    // Parameters for EL6 -> Serial Device
    fbSend: SendString;
    bSendBusy: BOOL;
    eLastSendErrorID: ComError_t;
    fbReceive: ReceiveString;
    sReceivedString: STRING;
    sLastReceivedString: STRING;
    bStringReceived: BOOL;
    bReceiveBusy: BOOL;
    bReceiveError: BOOL;
    eReceiveErrorID: ComError_t;
    bReceiveTimeout: BOOL;
    nReceiveCounter: UDINT;
    nSendCounter: UDINT;
    sStringToSend: STRING;
    fbFormatString: FB_FormatString;

    // Parameters for state-machine implementation
    nStep: INT := 0;
END_VAR

fbEL6Ctrl(
    Mode:= SERIALLINEMODE_EL6_22B,
    pComIn:= ADR(stIn_EL6),
    pComOut:= ADR(stOut_EL6),
    SizeComIn:= UINT_TO_INT(SIZEOF(stIn_EL6)),
    Error=> ,
    ErrorID=> eSerialLineErrorID,
    TxBuffer:= TxBuffer,
    RxBuffer:= RxBuffer );
IF fbEL6Ctrl.Error THEN
    bEL6CtrlError := TRUE;
    eEL6CtrlErrorID := fbEL6Ctrl.ErrorID;
END_IF
IF bSend THEN
    nStep := 10;
    bSend := FALSE;
    bDone := FALSE;
END_IF
// Attempt at solution that sends one command at a time, not on constant loop
CASE nStep OF
    0:
        ; // idle
    10:
        // Clear buffers in case any lingering data
        fbClearComBuffer(Buffer:=TxBuffer);
        fbClearComBuffer(Buffer:=RxBuffer);
        // Prepare string to send
        sStringToSend := CONCAT(sSendPrefix, CONCAT(sCmd, sSendSuffix));
        // Send string
        fbSend(	SendString:= sStringToSend,
                TXbuffer:= TxBuffer,
                Busy=> bSendBusy,
                Error=> eSendErrorID);
        IF fbSend.Error <> COMERROR_NOERROR THEN
            eLastSendErrorID := fbSend.Error;
        ELSE
            nSendCounter := nSendCounter + 1;
        END_IF
        nStep := nStep + 10;
    20:
        // Finish sending String
        IF fbSend.Busy THEN
            fbSend(	SendString:= sStringToSend,
                    TXbuffer:= TxBuffer,
                    Busy=> bSendBusy,
                    Error=> eSendErrorID);
            IF fbSend.Error <> COMERROR_NOERROR THEN
                eLastSendErrorID := fbSend.Error;
            ELSE
                nSendCounter := nSendCounter + 1;
            END_IF
        ELSE
            nStep := nStep + 10;
        END_IF
    30:
        // Get Reply
        fbReceive(
            Prefix:= sRecvPrefix,
            Suffix:= sRecvSuffix,
            Timeout:= tTimeout,
            ReceivedString:= sReceivedString,
            RXbuffer:= RxBuffer,
            StringReceived=> bStringReceived,
            Busy=> bReceiveBusy,
            Error=> eRecvErrorID,
            RxTimeout=> bReceiveTimeout );
        IF fbReceive.Error <> COMERROR_NOERROR THEN
            eReceiveErrorID := fbReceive.Error;
        END_IF
        IF bStringReceived THEN
            nReceiveCounter := nReceiveCounter + 1;
            // Check for response
            IF FIND(sReceivedString, sStringToSend)=0 THEN
                sResponse := sReceivedString;
                bDone := TRUE;
                nStep := 0;
            END_IF
        END_IF
END_CASE

END_FUNCTION_BLOCK

// POUs/Hardware/FB_GetPLCHostname
FUNCTION_BLOCK FB_GetPLCHostname
VAR_INPUT
    bEnable			: BOOL;
    tRetryDelay		: TIME := T#10s;
END_VAR
VAR_OUTPUT
    sHostname		: T_MaxString;
    bDone 			: BOOL;
    bError			: BOOL;
END_VAR
VAR
    fbGetHostName	: FB_GetHostName;

    tRetry 			: TON;
    bReset			: BOOL;
    bInitialized	: BOOL := FALSE;

END_VAR

IF bEnable THEN
    fbGetHostName.sNetID := '';

    IF NOT bInitialized OR (tRetry.Q AND NOT bDone) THEN
        bReset			:= TRUE;
        bInitialized	:= TRUE;
        fbGetHostName(bExecute:=FALSE);
    END_IF

    tRetry(IN:=bReset, PT:=tRetryDelay);

    bReset := FALSE;

    IF NOT bDone THEN
        fbGetHostName(bExecute:=TRUE, bError=>bError);
        IF NOT (fbGetHostName.bBusy OR bError) THEN
            sHostname	:= fbGetHostName.sHostName;
            bDone 		:= TRUE;
        END_IF
    END_IF
END_IF

END_FUNCTION_BLOCK

// POUs/Hardware/FB_GetPLCIPAddress
FUNCTION_BLOCK FB_GetPLCIPAddress
VAR_INPUT
    bEnable			: BOOL;
    tRetryDelay		: TIME := T#10s;
END_VAR
VAR_OUTPUT
    sIPAddress		: STRING(15);

    bDone 			: BOOL;
    bError			: BOOL;
END_VAR
VAR
    fbGetAdapterIP 	: FB_GetAdaptersInfo := (bExecute := TRUE, sNetID := ''); // Acquire IP of the correct adapter

    iIndex			: UDINT;

    tRetry 			: TON;
    bReset			: BOOL;
    bInitialized	: BOOL := FALSE;

END_VAR

IF bEnable THEN
    IF NOT bInitialized OR (tRetry.Q AND NOT bDone) THEN
        bReset			:= TRUE;
        bInitialized	:= TRUE;
        fbGetAdapterIP(bExecute:=FALSE);
    END_IF

    tRetry(IN:=bReset, PT:=tRetryDelay);
    bReset := FALSE;

    IF NOT bDone THEN
        fbGetAdapterIP(bExecute:=TRUE, bError=>bError);
        IF NOT (fbGetAdapterIP.bBusy or fbGetAdapterIP.bError) THEN
            FOR iIndex := 0 TO MAX_LOCAL_ADAPTERS DO
                IF FIND(fbGetAdapterIP.arrAdapters[iIndex].sIpAddr, GVL_Logger.sIpTidbit) <> 0 THEN
                    sIPAddress := fbGetAdapterIP.arrAdapters[iIndex].sIpAddr;
                    bDone := TRUE;
                    EXIT;
                END_IF
            END_FOR
        END_IF
    END_IF

END_IF

END_FUNCTION_BLOCK

// POUs/Hardware/FB_LED
FUNCTION_BLOCK FB_LED
(*
    Reads a percentage of illumination determined by the user and converts it to a raw value
    to send to the terminal output via the FB_AnalogOutput.

    The determination of the full scale raw value (FSV) is calculated via the iTermBits,
    which is setup as an input variable to be set according to the situation. This value
    is bounded by the FSV of the terminal set by the Beckhoff architecture: (2^15 - 1) = 32767.

    Through the configurable max raw value sent to the terminal output, this LED function block
    is applicable to a wider variety of hardware: whether it be simple Analog Voltage control,
    PWM voltage output, or current controlled output.

    As an initial application, this FB will be instituted for systems of vaccum chamber LED
    illuminators on TMO endstations, which are rated for 12 V max. They will be dimmed via the
    EL2502 terminal 24 V PWM output voltage control from 0-50% duty cycle.

    2022-5-03 Maarten Thomas-Bosum
*)
VAR_INPUT
    {attribute 'pytmc' := '
        pv: NAME
        io: io
        field: DESC Descriptive name for the LED
        autosave_pass0: VAL DESC
    '}
    ledName : STRING;

    iTermBits : UINT;

    {attribute 'pytmc' := '
        pv: ILL:PCT
        field: EGU %
    '}
    fIlluminatorPercent: LREAL;

    {attribute 'pytmc' := '
        pv: PWR
        field: ZNAM OFF
        field: ONAM ON
    '}
    bLedPower AT %Q*: BOOL;
END_VAR
VAR
    iIlluminatorINT AT %Q*: INT;
    fbSetIllPercent: FB_AnalogOutput;
END_VAR

// Illuminator conversion to percentage
fbSetIllPercent(
    fReal:=fIlluminatorPercent,
    fSafeMax:=100,
    fSafeMin:=0,
    iTermBits:=iTermBits,
    fTermMax:=100,
    fTermMin:=0,
    iRaw=>iIlluminatorINT);

IF  fIlluminatorPercent > 0 THEN
    bLedPower := TRUE;
ELSE
    bLEDPower := FALSE;
END_IF

END_FUNCTION_BLOCK

// POUs/Hardware/FB_TempSensor
FUNCTION_BLOCK FB_TempSensor
(*
    Handles scaling and default diagnostics for temperature sensors,
    such as thermocouples, RTDs, and others.
    2020-03-02 Zachary Lentz
*)
VAR_INPUT
    // Resolution parameter from the Beckhoff docs. Default is 0.1 for 0.1 degree resolution
    fResolution: LREAL := 0.1;
END_VAR
VAR_OUTPUT
    {attribute 'pytmc' := '
        pv: TEMP
        io: input
        field: EGU C
        field: PREC 2
    '}
    fTemp: LREAL;

    {attribute 'pytmc' := '
        pv: CONN
        io: input
        field: ONAM Connected
        field: ZNAM Disconnected
    '}
    bConnected: BOOL;

    {attribute 'pytmc' := '
        pv: ERR
        io: input
        field: ONAM True
        field: ZNAM False
    '}
    bError AT %I*: BOOL := TRUE;

    bUnderrange AT %I*: BOOL;
    bOverrange AT %I*: BOOL;
END_VAR
VAR
    iRaw AT %I*: INT;
END_VAR

// The manual states that we are disconnected if we are both overrange and in an error state
bConnected := NOT (bOverrange AND bError);
fTemp := INT_TO_LREAL(iRaw) * fResolution;

END_FUNCTION_BLOCK

// POUs/Hardware/FB_ThermoCouple
FUNCTION_BLOCK FB_ThermoCouple
(*
    Deprecated as of 2020-03-02, please use FB_TempSensor instead
    2019-10-09 Zachary Lentz
*)
{warning 'Function Block FB_ThermoCouple is deprecated and may be removed in a future release'}
VAR_INPUT
    // Ratio between raw value and actual temperature. Default is 10 for 10 steps per degree (or 0.1 degree resolution)
    iScale: INT := 10;
END_VAR
VAR_OUTPUT
    {attribute 'pytmc' := '
        pv: STC:TEMP
        io: input
    '}
    fTemp: LREAL;

    {attribute 'pytmc' := '
        pv: STC:CONN
        io: input
        field: ONAM Connected
        field: ZNAM Disconnected
    '}
    bConnected: BOOL;

    {attribute 'pytmc' := '
        pv: STC:ERR
        io: input
    '}
    bError AT %I*: BOOL;

    bUnderrange AT %I*: BOOL;
    bOverrange AT %I*: BOOL;
END_VAR
VAR
    iRaw AT %I*: INT;
END_VAR

// The manual states that we are disconnected if we are both overrange and in an error state
bConnected := NOT (bOverrange AND bError);
fTemp := INT_TO_LREAL(iRaw) / iScale;

END_FUNCTION_BLOCK

// POUs/Logger/F_SendUDPMessage
FUNCTION F_SendUDPMessage : HRESULT
VAR_INPUT
    sMessage			:	POINTER TO STRING;
    fbSocket			:	REFERENCE TO FB_ConnectionlessSocket;
    sHost				:	STRING;
    iPort				:	UINT;
END_VAR

VAR
    fbSend				:	FB_SocketUdpSendTo;
END_VAR

IF sMessage <> 0 AND __ISVALIDREF(fbSocket) THEN
    fbSend.hSocket		:= fbSocket.hSocket;
    fbSend.sRemoteHost	:= sHost;
    fbSend.nRemotePort	:= iPort;
    fbSend.pSrc 		:= sMessage;
    fbSend.cbLen		:= LEN2(sMessage);
    fbSend.bExecute	 	:= TRUE;
    fbSend();

    fbSend.bExecute 	R= fbSend.bBusy;
END_IF

END_FUNCTION

// POUs/Logger/FB_Listener
FUNCTION_BLOCK FB_Listener EXTENDS FB_ListenerBase
VAR_INPUT
END_VAR

VAR_OUTPUT
END_VAR

VAR
    nEventIdx			:	UINT := 0;
    nPendingEvents		:	UINT := 0;

    {attribute 'pytmc' := '
        pv: LogToVisualStudio
        io: io
    '}
    bLogToVisualStudio	:	BOOL := FALSE;

    {attribute 'pytmc' := '
        pv: MessagesSent
        io: i
    '}
    nCntMessagesSent 	: UDINT := 0;

    {attribute 'pytmc' := '
        pv: AlarmsRaised
        io: i
    '}
    nCntAlarmsRaised 	: UDINT := 0;

    {attribute 'pytmc' := '
        pv: AlarmsConfirmed
        io: i
    '}
    nCntAlarmsConfirmed : UDINT := 0;

    {attribute 'pytmc' := '
        pv: AlarmsCleared
        io: i
    '}
    nCntAlarmsCleared 	: UDINT := 0;

    {attribute 'pytmc' := '
        pv: MinSeverity
        io: io
    '}
    eMinSeverity	 	: TcEventSeverity;

    {attribute 'analysis' := '-33'}
    {attribute 'pytmc' := '
        pv: Log
    '}
    stEventInfo 		:	REFERENCE TO ST_LoggingEventInfo;

    stPendingEvents		:	ARRAY [0..nMaxEvents - 1] OF ST_PendingEvent;
    ipMessageConfig		:	ITcEventFilterConfig;
    fbSocket			:	POINTER TO FB_ConnectionlessSocket;
    bConfigured			:	BOOL	:= FALSE;


END_VAR

VAR_IN_OUT

END_VAR

VAR CONSTANT
    // The maximum number of events allowed *per-cycle*
    nMaxEvents			:	UINT := 10;
END_VAR

(*
    Configure an event class + severity
*)
METHOD Configure : HRESULT
VAR_INPUT
    i_EventClass 	:	GUID;
    i_MinSeverity	:	TcEventSeverity := TcEventSeverity.Verbose;
    i_fbSocket		:	POINTER TO FB_ConnectionlessSocket;
END_VAR

VAR_INST
    bSubscribed		:	BOOL := FALSE;
END_VAR
IF bSubscribed THEN
    Unsubscribe();
END_IF

THIS^.Subscribe(ADR(ipMessageConfig), 0);
bSubscribed 	:= TRUE;
eMinSeverity 	:= i_MinSeverity;
fbSocket	  	:= i_fbSocket;

IF (ipMessageConfig = 0) THEN
    Configure 	:= 1;
    bConfigured := FALSE;
ELSE
    ipMessageConfig.AddEventClass(i_EventClass, i_MinSeverity);
    Configure 	:= 0;
    bConfigured := TRUE;
END_IF
END_METHOD

{attribute 'analysis' := '-33'}
PROPERTY PUBLIC LogToVisualStudio : BOOL
GET
LogToVisualStudio := bLogToVisualStudio;
END_GET
SET
VAR
    bValue : BOOL;
END_VAR
THIS^.bLogToVisualStudio := bValue;
END_SET
END_PROPERTY

METHOD OnAlarmCleared
VAR_INPUT
    fbEvent : REFERENCE TO FB_TcEvent;
END_VAR
(* Callback run from THIS^.Execute() *)
nCntAlarmsCleared := nCntAlarmsCleared + 1;
StoreEvent(fbEvent, eEventType:=E_LogEventType.AlarmCleared);
END_METHOD

METHOD OnAlarmConfirmed
VAR_INPUT
    fbEvent : REFERENCE TO FB_TcEvent;
END_VAR
(* Callback run from THIS^.Execute() *)
nCntAlarmsConfirmed := nCntAlarmsConfirmed + 1;
StoreEvent(fbEvent, eEventType:=E_LogEventType.AlarmConfirmed);
END_METHOD

METHOD OnAlarmRaised
VAR_INPUT
    fbEvent : REFERENCE TO FB_TcEvent;
END_VAR
(* Callback run from THIS^.Execute() *)
nCntAlarmsRaised := nCntAlarmsRaised + 1;
StoreEvent(fbEvent, eEventType:=E_LogEventType.AlarmRaised);
END_METHOD

METHOD OnMessageSent
VAR_INPUT
    fbEvent : REFERENCE TO FB_TcEvent;
END_VAR
(* Callback run from THIS^.Execute() *)
nCntMessagesSent := nCntMessagesSent + 1;
StoreEvent(fbEvent, eEventType:=E_LogEventType.MessageSent);
END_METHOD

METHOD PublishEvents : HRESULT
VAR
    nEvent				:	UINT;
    stPendingEvent		:	REFERENCE TO ST_PendingEvent;
    stEventInfo			:	REFERENCE TO ST_LoggingEventInfo;
    fbRequestEventText	:	REFERENCE TO FB_RequestEventText;
END_VAR

VAR_INST
    fbJson				:	FB_JsonSaxWriter;
    fbJsonDataType		:	FB_JsonReadWriteDataType;
    sJsonDoc			:	STRING(10000);

END_VAR

IF nPendingEvents = 0 THEN
    RETURN;
END_IF

FOR nEvent := 0 TO nMaxEvents - 1 DO
    stPendingEvent REF= stPendingEvents[nEvent];
    IF NOT stPendingEvent.bInUse THEN
        CONTINUE;
    END_IF

    fbRequestEventText REF= stPendingEvent.fbRequestEventText;
    stEventInfo 	   REF= stPendingEvent.stEventInfo;

    IF fbRequestEventText.bError THEN
        stEventInfo.Msg := '(Unable to retrieve message)';
    ELSIF NOT fbRequestEventText.bBusy THEN
        fbRequestEventText.GetString(stEventInfo.msg, SIZEOF(stEventInfo.msg));
    ELSE
        CONTINUE;
    END_IF

    IF bConfigured THEN
        stEventInfo.plc := GVL_Logger.sPlcHostname;

        // Generate the JSON message
        fbJson.ResetDocument();
        fbJsonDataType.AddJsonValueFromSymbol(fbJson, 'ST_LoggingEventInfo', SIZEOF(stEventInfo), ADR(stEventInfo));
        fbJson.CopyDocument(sJsonDoc, SIZEOF(sJsonDoc));

        SendMessage(sMessage:=ADR(sJsonDoc));
    END_IF

    // Mark as not in use, and fill in this event in the next StoreEvent call
    nPendingEvents			:= nPendingEvents - 1;
    stPendingEvent.bInUse 	:= FALSE;
    nEventIdx 				:= nEvent;

END_FOR
END_METHOD

METHOD SendMessage : HRESULT
VAR_INPUT
    sMessage		:	POINTER TO STRING;
END_VAR

VAR
    sLogStr			:	T_MaxString;
END_VAR
(* For subclasses to override, if necessary *)
IF sMessage = 0 THEN
    RETURN;
END_IF

// Optionally log it to Visual Studio's message list
IF bLogToVisualStudio THEN
     // Keep the message length under 255 (extended string function for LEFT/MID do not exist)
    STRNCPY(ADR(sLogStr), sMessage, MIN(220, SIZEOF(sLogStr)));
    ADSLOGSTR(
        msgCtrlMask := ADSLOG_MSGTYPE_HINT,
        msgFmtStr   := '[Logger JSON Debug] %s',
        strArg      := sLogStr
    );
END_IF

IF fbSocket <> 0 THEN
    // And send it along to logstash
    F_SendUDPMessage(sMessage:=sMessage, fbSocket:=fbSocket^,
                     sHost:=GVL_Logger.cLogHost, iPort:=GVL_Logger.iLogPort);
END_IF
END_METHOD

METHOD PRIVATE StoreEvent : HRESULT
VAR_INPUT
    fbEvent		:	REFERENCE TO FB_TcEvent;
    eEventType	:	E_LogEventType;
END_VAR

VAR
    stPendingEvent	:	REFERENCE TO ST_PendingEvent;
    stEventInfo		:	REFERENCE TO ST_LoggingEventInfo;
    nFailures		:	UINT := 0;
END_VAR
IF fbEvent.eSeverity < eMinSeverity THEN
    // Ignore all messages below the minimum severity
    RETURN;
ELSIF NOT __ISVALIDREF(fbEvent) THEN
    RETURN;
END_IF

// Find the next slot to use in stPendingEvents
WHILE stPendingEvents[nEventIdx].bInUse AND nFailures < nMaxEvents DO
    nFailures := nFailures + 1;
    IF ((nEventIdx := (nEventIdx + 1)) = nMaxEvents) THEN
        nEventIdx := 0;
    END_IF
END_WHILE

IF (nFailures = nMaxEvents) THEN
    ADSLOGSTR(
        msgCtrlMask := ADSLOG_MSGTYPE_ERROR,
        msgFmtStr   := 'Logging message buffer full (%s)',
        strArg		:= UINT_TO_STRING(nMaxEvents),
    );
    RETURN;
END_IF

nPendingEvents			:=	nPendingEvents + 1;
nCntMessagesSent 		:=	nCntMessagesSent + 1;

stPendingEvent			REF= stPendingEvents[nEventIdx];
stEventInfo 			REF= stPendingEvent.stEventInfo;
stPendingEvent.bInUse 	:= TRUE;

stEventInfo.id 			:= fbEvent.nEventId;
stEventInfo.event_class	:= GUID_TO_STRING(fbEvent.EventClass);
stEventInfo.severity 	:= fbEvent.eSeverity;
stEventInfo.ts			:= F_ConvertTicksToUnixTimestamp(fbEvent.nTimestamp);
stEventInfo.source 		:= fbEvent.ipSourceInfo.sName;
stEventInfo.event_type	:= eEventType;

fbEvent.GetJsonAttribute(stEventInfo.json, SIZEOF(stEventInfo.json));
stPendingEvent.fbRequestEventText.Request(eventClass:=fbEvent.EventClass, nEventId:=fbEvent.nEventId, nLangId:=1033, ipArgs:=fbEvent.ipArguments);
END_METHOD

END_FUNCTION_BLOCK

// POUs/Logger/FB_LogHandler
FUNCTION_BLOCK FB_LogHandler
VAR_INPUT

    {attribute 'pytmc' := '
        pv: ADS
    '}
    fbTcAdsListener : FB_Listener;

    {attribute 'pytmc' := '
        pv: Router
    '}
    fbTcRouterListener : FB_Listener;

    {attribute 'pytmc' := '
        pv: RTime
    '}
    fbTcRTimeListener : FB_Listener;

    {attribute 'pytmc' := '
        pv: System
    '}
    fbTcSystemListener : FB_Listener;

    {attribute 'pytmc' := '
        pv: Windows
    '}
    fbWindowsListener : FB_Listener;

    {attribute 'pytmc' := '
        pv: LCLS
    '}
    fbLCLSListener 	: FB_Listener;

END_VAR
VAR_OUTPUT
END_VAR

VAR

    bInitialized	:	BOOL	:= FALSE;
    bReadyToLog		: 	BOOL	:= FALSE;
    rtFirstLog		: 	R_TRIG;

    fbGetHostName 	: FB_GetPLCHostname;
    fbGetIP		 	: FB_GetPLCIPAddress;

    fbListener		:	REFERENCE TO FB_Listener;
    fbListeners		: 	ARRAY [0..nNumListeners - 1] OF POINTER TO FB_Listener;

    // Default minimum severity for subscriptions
    eMinSeverity	:	TcEventSeverity := TcEventSeverity.Verbose;

    {attribute 'naming' := 'omit'}
    rtReset				:	R_TRIG; //Reset trigger
    bReset				:	BOOL;

    fbSocket	   		:	FB_ConnectionlessSocket;

    nI					:	UINT;

    SocketEnable : BOOL;

    ctuSocketError : CTU := (PV:=3); // Circuit breaker for socket errors. 3 errors before it stops.

    tRetryConnection : TON := (PT:=T#1h); // Retry after an hour

    tofTrickleBreakerPre : TOF := (PT:=T#1s);
    tonTrickleBreaker : TON := (PT := GVL_Logger.nTrickleTripTime);
    bTripCon : BOOL;
END_VAR

VAR CONSTANT
    nNumListeners		:	UINT	:= 6;
END_VAR

IF NOT bInitialized THEN
    bInitialized := TRUE;
    fbTcAdsListener.Configure(i_EventClass:=TC_EVENT_CLASSES.TcGeneralAdsEventClass, i_MinSeverity:=eMinSeverity, i_fbSocket:=ADR(fbSocket));
    fbTcRouterListener.Configure(i_EventClass:=TC_EVENT_CLASSES.TcRouterEventClass, i_MinSeverity:=eMinSeverity, i_fbSocket:=ADR(fbSocket));
    fbTcRTimeListener.Configure(i_EventClass:=TC_EVENT_CLASSES.TcRTimeEventClass, i_MinSeverity:=eMinSeverity, i_fbSocket:=ADR(fbSocket));
    fbTcSystemListener.Configure(i_EventClass:=TC_EVENT_CLASSES.TcSystemEventClass, i_MinSeverity:=eMinSeverity, i_fbSocket:=ADR(fbSocket));
    fbWindowsListener.Configure(i_EventClass:=TC_EVENT_CLASSES.Win32EventClass, i_MinSeverity:=eMinSeverity, i_fbSocket:=ADR(fbSocket));
    fbLCLSListener.Configure(i_EventClass:=TC_EVENT_CLASSES.LCLSGeneralEventClass, i_MinSeverity:=eMinSeverity, i_fbSocket:=ADR(fbSocket));

    fbListeners[0] := ADR(fbTcAdsListener);
    fbListeners[1] := ADR(fbTcRouterListener);
    fbListeners[2] := ADR(fbTcRTimeListener);
    fbListeners[3] := ADR(fbTcSystemListener);
    fbListeners[4] := ADR(fbWindowsListener);
    fbListeners[5] := ADR(fbLCLSListener);

END_IF

fbGetHostName(
    bEnable := TRUE,
    sHostname => GVL_Logger.sPlcHostname,
);

fbGetIP(
    bEnable := TRUE,
    sIPAddress => fbSocket.sLocalHost
);

(* Ensure the socket is ready for when JSON documents are emitted *)
rtReset(CLK:=bReset);

IF (rtReset.Q AND fbSocket.bEnable) THEN
    fbSocket(bEnable:=FALSE);
END_IF

// Disable fbSocket if too many errors occur
ctuSocketError(CU:=fbSocket.bError, RESET:=tRetryConnection.Q OR rtReset.Q);
SocketEnable R= ctuSocketError.Q;
// Retry an hour later
tRetryConnection(IN:=ctuSocketError.Q);
SocketEnable S= tRetryConnection.Q OR rtReset.Q;

fbSocket(
    nLocalPort:=0,
    bEnable:=fbGetIP.bDone,
    nMode:=CONNECT_MODE_ENABLEDBG,
);

bReadyToLog := (
    fbGetHostName.bDone AND
    fbGetIP.bDone AND
    bInitialized AND
    fbSocket.bEnable AND
    NOT fbSocket.bError AND
    fbSocket.eState = E_SocketConnectionlessState.eSOCKET_CREATED
);
rtFirstLog(CLK:=bReadyToLog);

IF rtFirstLog.Q THEN
    fbRootLogger(sMsg:='Logging system online', eSevr:=TcEventSeverity.Info,
                 eSubsystem:=E_Subsystem.NILVALUE);
END_IF

CircuitBreaker();

(* Poke all of the listeners *)
FOR nI := 0 TO nNumListeners - 1 DO
    fbListener REF= fbListeners[nI]^;
    fbListener.Execute();
    fbListener.PublishEvents();
END_FOR

ACTION CircuitBreaker:
// Global log circuit breaker
(*
Logic explanation
We want to trip if there is a constant stream of messages being emitted by this PLC. We also
only want the noisy offenders to trip. To target them we set a global trickle tripped flag
using this logic here. Then each individual FB_LogMessage evaluates itself to see if it's
sending a message too frequently (ie. it's being called to often).

This logic is attempting to implement the following:
1. Trip if the total events exceeds the nTrickleThreshold for >10s
2. Sustain the timer if the event count drops for a handful of cycles since usually a cycle amounts to 10ms, losing a few
should not stop the trickle timer.
*)
bTripCon := GVL_Logger.nGlobAccEvents >0;

tofTrickleBreakerPre(IN:=bTripCon);
tonTrickleBreaker(IN:=tofTrickleBreakerPre.Q);

GVL_Logger.bTrickleTripped S= tonTrickleBreaker.Q AND bTripCon;

GVL_Logger.nGlobAccEvents := 0; // reset the count for the next cycle
END_ACTION

END_FUNCTION_BLOCK

// POUs/Logger/SYSTEM_TIME_TO_RFC3339
//Converts Beckhoff PLC SYSTEMTIME to RFC3339 time format as a string
{attribute 'naming' := 'omit'}
{attribute 'analysis' := '-23'}
FUNCTION SYSTEM_TIME_TO_RFC3339 : STRING(255)
VAR_INPUT
    {attribute 'naming' := 'omit'}
    tCurrentTime	:	TIMESTRUCT; //TIMESTRUCT Time to convert to RFC3339
END_VAR
VAR
END_VAR

SYSTEM_TIME_TO_RFC3339 := CONCAT(REPLACE(SYSTEMTIME_TO_STRING(tCurrentTime), 'T', 1, 11), 'Z');

END_FUNCTION

// POUs/Tests/FB_CircuitBreaker_Test
{attribute 'call_after_init'}
FUNCTION_BLOCK FB_CircuitBreaker_Test EXTENDS TcUnit.FB_TestSuite
VAR_INPUT
END_VAR
VAR_OUTPUT
END_VAR
VAR
END_VAR

AutoReset();
SingleBadLogger();
DeathByManySmall();

METHOD AutoReset
VAR_INPUT
END_VAR
VAR_INST
    fbLog : FB_LogMessage := (
        bEnableAutoReset:=TRUE,
        nTripResetPeriod := T#5s);

    //Auto reset test
    tonAutoResetTest : TON;

    {attribute 'analysis' := '-27'}
    Init : BOOL := TRUE;
END_VAR
(* Test that the CB resets itself after a cooldown period *)
TEST('AutoReset');
IF Init THEN
    fbLog.CircuitBreaker();
    WRITE_PROTECTED_BOOL(ADR(fbLog.bTripped), TRUE);
    WRITE_PROTECTED_BOOL(ADR(fbLog.bLocalTripped), TRUE);
    fbLog.CircuitBreaker();
    fbLog.CircuitBreaker();
    Init := FALSE;
END_IF

tonAutoResetTest(IN:=NOT Init, PT:=T#6s);

IF tonAutoResetTest.Q THEN

    fbLog.CircuitBreaker();

    AssertFalse(fbLog.bTripped,
        'Circuit breaker should be reset automatically');

    TEST_FINISHED_NAMED('AutoReset');
END_IF
END_METHOD

METHOD DeathByManySmall
VAR_INPUT
END_VAR
VAR

END_VAR
VAR_INST
    fbLogNoisy : FB_LogMessage;
    tNoisy : TON := (PT:=T#50ms); //50ms is > the local trip threshold default of 1ms
    fbLogNice : FB_LogMessage := (nTrickleTripThreshold:=T#2s);
    tNice : TON := (PT:=T#5s);
    tTrickle : TON := (PT:= GVL_Logger.nTrickleTripTime + T#1s);
    fbLogHandler : FB_LogHandler;
END_VAR
TEST('ManySmall');
// Create a condition where
// a few loggers did their thing, while keeping under the
// local logging rate limit until the global trickle trip
// was triggered. Then verify only those loggers that
// were just a little too noisy, would trip off, while others stayed up.

fbLogHandler.CircuitBreaker();

// Call this guy every 50ms or so.
tNoisy(IN := NOT tNoisy.Q);
IF tNoisy.Q THEN
    fbLogNoisy.CircuitBreaker();
END_IF

// Call this guy every 5s or so
tNice(IN := NOT tNoisy.Q);
IF tNice.Q THEN
    fbLogNice.CircuitBreaker();
END_IF

tTrickle(IN:=TRUE);
IF tTrickle.Q THEN
    AssertTrue(fbLogNoisy.bLocalTrickleTripped AND NOT fbLogNice.bLocalTrickleTripped,
            'Only Noisy should be tripped.');
    TEST_FINISHED_NAMED('ManySmall');
END_IF
END_METHOD

METHOD SingleBadLogger
VAR_INPUT
END_VAR
VAR
    idx : UINT;
END_VAR
VAR_INST
    fbLog : FB_LogMessage := (
        bEnableAutoReset:=TRUE,
        nTripResetPeriod := T#5s);
END_VAR
ResetCircuitBreakerGlobals();

(* In this scenario, a logger trips off because it has been called too many times
in one cycle, leading to a large excess of messages.
*)
TEST('LocalFastTrip');
    FOR idx := 0 TO GVL_LOGGER.nMinTimeViolationAcceptable + 1 DO
        fbLog.CircuitBreaker();
    END_FOR

    AssertTrue(fbLog.bLocalTripped AND NOT fbLog.bLocalTrickleTripped,
        'Only local trip should occur in these conditions');
TEST_FINISHED();
END_METHOD

END_FUNCTION_BLOCK

// POUs/Tests/ResetCircuitBreakerGlobals
FUNCTION ResetCircuitBreakerGlobals : BOOL
VAR_INPUT
END_VAR
VAR
END_VAR

GVL_Logger.bTrickleTripped := FALSE;
GVL_Logger.nGlobAccEvents := 0;

END_FUNCTION

// POUs/Tests/FB_ECATAutoRestart_Test

FUNCTION_BLOCK FB_ECATAutoRestart_Test EXTENDS TcUnit.FB_TestSuite
VAR
    fbECATAutoRestart : FB_ECATAutoRestart;

    fbTON_TestTimer		: TON;
    bStartTest			: BOOL := FALSE;


END_VAR


TestSingleLogPerTransitionExpect4Logs();
TestAnyStateExpectChangeToOpStateInSeq();
TestNotEnabledExpectNoStateChange();
Test5RetriesExpectErrorStopTrying();
TestBadAddressExpectError();


METHOD Test5RetriesExpectErrorStopTrying
VAR_INPUT
END_VAR
VAR
    nIndex                  : INT;
    nStateMachineState      : INT;

    // State Machine Control Inputs
    bEnable                 : BOOL;
    bfbGetBusy              : BOOL;
    bfbGetError              : BOOL;
    nCurretState            : WORD;
    bfbSetBusy              : BOOL;
    bfbSetError             : BOOL;

    // State Machine Control Outputs
    bfbGetUpdatedState      : BOOL;
    bSetNextState           : BOOL;
    nNextState              : WORD;
    sLogMessage             : T_MaxString;
    bLog                    : BOOL;

END_VAR

TEST('Test5RetriesExpectErrorStopTrying');

nStateMachineState := 1; // Start Test on Start State
bEnable := TRUE;
bfbGetBusy := FALSE;
bfbGetError := FALSE;
nCurretState := EC_DEVICE_STATE_PREOP;
bfbSetBusy := FALSE;
bfbSetError := TRUE;

FOR nIndex := 1 TO 20 DO
    fbECATAutoRestart.StateMachine(bEnable:=bEnable,
        bfbGetBusy := bfbGetBusy,
        bfbGetError := bfbGetError,
        bfbGetUpdatedState => bfbGetUpdatedState,
        nCurretState := nCurretState,
        nNextState => nNextState,
        sLogMessage=> sLogMessage,
        bLog=> bLog,
        bSetNextState=> bSetNextState,
        bfbSetBusy := bfbSetBusy,
        bfbSetError := bfbSetError);
END_FOR


AssertEquals_BOOL(Expected:=TRUE,
                    Actual:= fbECATAutoRestart.bStopTrying,
                    Message:='bStopTrying was not set after trying to get new position after 20 Cycles');

// CLEAR ANY ERRORS AFTER TESTS
FOR nIndex := 1 TO 3 DO
    fbECATAutoRestart.StateMachine(bEnable:=FALSE,
        bfbGetBusy := bfbGetBusy,
        bfbGetError := bfbGetError,
        bfbGetUpdatedState => bfbGetUpdatedState,
        nCurretState := nCurretState,
        nNextState => nNextState,
        sLogMessage=> sLogMessage,
        bLog=> bLog,
        bSetNextState=> bSetNextState,
        bfbSetBusy := bfbSetBusy,
        bfbSetError := bfbSetError);
END_FOR

TEST_FINISHED();
END_METHOD


METHOD TestAnyStateExpectChangeToOpStateInSeq
VAR_INPUT
END_VAR
VAR

    // State Machine Control Inputs
    bEnable                 : BOOL;
    bfbGetBusy              : BOOL;
    bfbGetError				: BOOL;
    nCurretState            : WORD;
    bfbSetBusy              : BOOL;
    bfbSetError             : BOOL;

    // State Machine Control Outputs
    bfbGetUpdatedState      : BOOL;
    bSetNextState           : BOOL;
    nNextState              : WORD;
    sLogMessage             : T_MaxString;
    bLog                    : BOOL;
    // TestAnyStateChangeOpInSeq Vars

    nIndex          : INT := 1;
    aPossibleStart : ARRAY [1 .. 4] OF BYTE := [EC_DEVICE_STATE_BOOTSTRAP,
                                                EC_DEVICE_STATE_INIT,
                                                EC_DEVICE_STATE_PREOP,
                                                EC_DEVICE_STATE_SAFEOP];
    nStartIndex : INT := 0;


END_VAR

TEST('TestAnyStateExpectChangeToOpStateInSeq');


bEnable := TRUE;
bfbGetBusy := FALSE;
bfbSetBusy := FALSE;
bfbSetError := FALSE;
bfbGetError := FALSE;




FOR nStartIndex := 1 TO 4 DO
    nCurretState := aPossibleStart[nStartIndex];
    // Takes 3 cycles for statemachine to update state
    // 4 - nStartIndex is number of steps needed to return to OP
    FOR nIndex := 1 TO 3 * 4 - nStartIndex DO
    fbECATAutoRestart.StateMachine
            (bEnable:=bEnable,
            bfbGetBusy := bfbGetBusy,
            bfbGetError := bfbGetError,
            bfbGetUpdatedState => bfbGetUpdatedState,
            nCurretState := nCurretState,
            nNextState => nNextState,
            sLogMessage=> sLogMessage,
            bLog=> bLog,
            bSetNextState=> bSetNextState,
            bfbSetBusy := bfbSetBusy,
            bfbSetError := bfbSetError);

    IF bSetNextState THEN
        nCurretState := nNextState;
    END_IF
    END_FOR

    AssertEquals_BYTE(Expected:=EC_DEVICE_STATE_OP,
        Actual:= TO_BYTE(nCurretState),
        Message:='Test Did not Return to OP');
END_FOR

 TEST_FINISHED();
END_METHOD


METHOD TestBadAddressExpectError
VAR_INPUT
END_VAR
VAR
    bError				: BOOL;
    bErrorId			: UDINT;
    nIndex				: INT;
END_VAR

TEST('TestBadAddressExpectError');

FOR nIndex := 1 TO 6 DO

    fbECATAutoRestart(sNetId:='1.0.0.0.1',
                    nSlaveAddr:=11101,
                    bEnable:= TRUE,
                    bError=>bError,
                    nErrorId=>bErrorId);


    IF bError THEN
    AssertEquals_BOOL(Expected:=TRUE,
        Actual:=bError,
        Message:= 'Expected bError to be TRUE');

    AssertEquals_UDINT(Expected:= 7,
        Actual:= bErrorId,
        Message:= 'Expected ERR_TARGETMACHINENOTFOUND (0x7)');

    END_IF
END_FOR

   TEST_FINISHED();
END_METHOD


METHOD TestNotEnabledExpectNoStateChange
VAR_INPUT
END_VAR
VAR
    nStateMachineStartState      : INT;
    // State Machine Control Inputs
    bEnable                 : BOOL;
    bfbGetBusy              : BOOL;
    bfbGetError				: BOOL;
    nCurretState            : WORD;
    bfbSetBusy              : BOOL;
    bfbSetError             : BOOL;

    // State Machine Control Outputs
    bfbGetUpdatedState      : BOOL;
    bSetNextState           : BOOL;
    nNextState              : WORD;
    sLogMessage             : T_MaxString;
    bLog                    : BOOL;

END_VAR

TEST('TestNotEnabledExpectNoStateChange');

nStateMachineStartState := 1;
bEnable := FALSE;
bfbGetBusy := FALSE;
nCurretState := EC_DEVICE_STATE_PREOP;
bfbSetBusy := FALSE;
bfbSetError := TRUE;
bfbGetError := FALSE;

fbECATAutoRestart.StateMachine(bEnable:=bEnable,
    bfbGetBusy := bfbGetBusy,
    bfbGetError	:= bfbGetError,
    bfbGetUpdatedState => bfbGetUpdatedState,
    nCurretState := nCurretState,
    nNextState => nNextState,
    sLogMessage=> sLogMessage,
    bLog=> bLog,
    bSetNextState=> bSetNextState,
    bfbSetBusy := bfbSetBusy,
    bfbSetError := bfbSetError);


AssertEquals_WORD(Expected:= 0,
                    Actual:= nNextState,
                    Message:= 'When bEnable is False, nNextState should not return anything');

TEST_FINISHED();
END_METHOD

METHOD TestSingleLogPerTransitionExpect4Logs
VAR_INPUT
END_VAR

VAR
        // State Machine Control Inputs
    bEnable                 : BOOL;
    bfbGetBusy              : BOOL;
    nCurretState            : WORD;
    bfbSetBusy              : BOOL;
    bfbSetError             : BOOL;
    bfbGetError				: BOOL;

    // State Machine Control Outputs
    bfbGetUpdatedState      : BOOL;
    bSetNextState           : BOOL;
    nNextState              : WORD;
    sLogMessage             : T_MaxString;
    bLog                    : BOOL;

    nIndex          : INT := 1;
    nLogCount       : INT := 0;
END_VAR

TEST('TestSingleLogPerTransitionExpect4Logs');

fbTON_TestTimer(IN:=bStartTest,PT:=T#1s);
IF  NOT bStartTest THEN bStartTest := TRUE; END_IF

bEnable := TRUE;
bfbGetBusy := FALSE;
bfbSetBusy := FALSE;
bfbSetError := FALSE;
bfbGetError := FALSE;

nCurretState := EC_DEVICE_STATE_INIT;
// Using More cyles then needed
 FOR nIndex := 1 TO 3 * 4 DO
    fbECATAutoRestart.StateMachine
            (bEnable:=bEnable,
            bfbGetBusy := bfbGetBusy,
            bfbGetError := bfbGetError,
            bfbGetUpdatedState => bfbGetUpdatedState,
            nCurretState := nCurretState,
            nNextState => nNextState,
            sLogMessage=> sLogMessage,
            bLog=> bLog,
            bSetNextState=> bSetNextState,
            bfbSetBusy := bfbSetBusy,
            bfbSetError := bfbSetError);

    IF bLog THEN
        nLogCount := nLogCount + 1;
    END_IF
END_FOR

AssertEquals_INT(Expected:= 4,
    Actual:=nLogCount,
    Message:='More than 4 Logs where Produced');

TEST_FINISHED();
END_METHOD

END_FUNCTION_BLOCK

// POUs/Tests/FB_FlutterDetection_Test
FUNCTION_BLOCK FB_FlutterDetection_Test EXTENDS TcUnit.FB_TestSuite
VAR_INPUT
END_VAR
VAR_OUTPUT
END_VAR
VAR
    fbFlutterDet : FB_FlutterDetection;

    nFirstCycleCount : UDINT;
    nCurrentSystemCycle : UDINT;
    nCurrentLocalCycle : UDINT;
END_VAR

TestFlutterResolution();
TestFlutterReset();

METHOD TestFlutterReset
VAR_INST
    fbTestTimer : TON := (PT := T#300ms);
    bInit : BOOL := FALSE;
    bVarToMonitor : BOOL := TRUE;
END_VAR
(* after trip, function should latch exceeded flag remains tripped. Finally,
check that after reset, the coount resets and the exceeded flag
goes low, then trips again. *)
TEST('TestFlutterReset');
IF NOT bInit THEN
    nFirstCycleCount := _TaskInfo[GETCURTASKINDEXEX()].CycleCount;
    bInit := TRUE;
END_IF
nCurrentSystemCycle := _TaskInfo[GETCURTASKINDEXEX()].CycleCount;
nCurrentLocalCycle := nCurrentSystemCycle - nFirstCycleCount;
fbTestTimer(IN := TRUE);
bVarToMonitor := NOT bVarToMonitor;

fbFlutterDet(bVarToMonitor:=bVarToMonitor ,fPastTime:=T#50ms ,nMaxFlipsAllowed:=4);

CASE nCurrentLocalCycle OF
10:
    AssertTrue(fbFlutterDet.bExceededFlipMax, 'exceeded flag not present');
11:
    // latched
    AssertTrue(fbFlutterDet.bExceededFlipMax, 'exceeded flag not present');
12:
    // latched
    AssertTrue(fbFlutterDet.bExceededFlipMax, 'exceeded flag not present');
    fbFlutterDet(bReset:=TRUE);
13:
    // reset
    AssertFalse(fbFlutterDet.bExceededFlipMax, 'false exceeded');
25:
    // lose a few cycles on reset.
    AssertTrue(fbFlutterDet.bExceededFlipMax, 'exceeded flag not present');
END_CASE

IF fbTestTimer.Q THEN
    TEST_FINISHED();
END_IF
END_METHOD

METHOD TestFlutterResolution
VAR_INST
    fbTestTimer : TON := (PT := T#200ms);

    fbFlutterDetExceedResolution : FB_FlutterDetection;
    fbFlutterDetMaxResolution : FB_FlutterDetection;
    nCycleTime : UDINT;
    nCalcCycleTime : TIME;
    nNumCycles : UDINT := 4;
    bVarToMonitor : BOOL := TRUE;
END_VAR
(*Test the max flips that can be detected, should be number of cycles - 1*)

TEST('TestFlutterResolution');
fbTestTimer(IN := TRUE);

nCycleTime := _TaskInfo[GETCURTASKINDEXEX()].CycleTime;
nCycleTime := nCycleTime / 10000; //convert to ms
nCalcCycleTime := UDINT_TO_TIME(nCycleTime * nNumCycles);

fbFlutterDetExceedResolution(bVarToMonitor:=bVarToMonitor, fPastTime:=nCalcCycleTime, nMaxFlipsAllowed:=nNumCycles);
fbFlutterDetMaxResolution(bVarToMonitor:=bVarToMonitor, fPastTime:=nCalcCycleTime, nMaxFlipsAllowed:=nNumCycles - 1);
bVarToMonitor := NOT bVarToMonitor;

IF fbTestTimer.Q THEN
    assertFalse(fbFlutterDetExceedResolution.bExceededFlipMax,'Flutter shouldnt be detected');
    assertTrue(fbFlutterDetMaxResolution.bExceededFlipMax,'Flutter not detected');
    TEST_FINISHED();
END_IF
END_METHOD

END_FUNCTION_BLOCK

// POUs/Tests/FB_Test_EpicsCentroidMonitor
{attribute 'call_after_init'}
FUNCTION_BLOCK FB_Test_EpicsCentroidMonitor EXTENDS TcUnit.FB_TestSuite
VAR_INPUT
END_VAR
VAR_OUTPUT
END_VAR
VAR
END_VAR

TestBasics();

METHOD TestBasics
VAR_INPUT
END_VAR
VAR_INST
    fbMonitor : FB_EpicsCentroidMonitor;
    nCount : INT := 0;
END_VAR
TEST('Basic');

nCount := 0;

nCount := nCount + 1;
WriteCentroidValue(fbMonitor:=fbMonitor, fX:=0.0, fY:=0.0, nCount:=nCount, nX_Severity:=0, nY_Severity:=0, nCount_Severity:=0, tLastUpdate:=T#0S);
fbMonitor();

nCount := nCount + 1;
WriteCentroidValue(fbMonitor:=fbMonitor, fX:=0.1, fY:=0.1, nCount:=nCount, nX_Severity:=0, nY_Severity:=0, nCount_Severity:=0, tLastUpdate:=T#0S);
fbMonitor(fMinimumValidChange:=0.0);

AssertTrue(fbMonitor.bIsUpdating, Message:='Centroid not reporting updating');

TEST_FINISHED();

TEST('Min change');

nCount := nCount + 1;
WriteCentroidValue(fbMonitor:=fbMonitor, fX:=0.0, fY:=0.0, nCount:=nCount, nX_Severity:=0, nY_Severity:=0, nCount_Severity:=0, tLastUpdate:=T#0S);
fbMonitor(fMinimumValidChange:=0.1, fMaximumFrameTime:=0.2);

nCount := nCount + 1;
WriteCentroidValue(fbMonitor:=fbMonitor, fX:=0.05, fY:=0.05, nCount:=nCount, nX_Severity:=0, nY_Severity:=0, nCount_Severity:=0, tLastUpdate:=T#0.1S);
fbMonitor(fMinimumValidChange:=0.1, fMaximumFrameTime:=0.2);
AssertFalse(fbMonitor.bIsUpdating, Message:='Centroid update below threshold and is not updating');

nCount := nCount + 1;
WriteCentroidValue(fbMonitor:=fbMonitor, fX:=0.5, fY:=0.5, nCount:=nCount, nX_Severity:=0, nY_Severity:=0, nCount_Severity:=0, tLastUpdate:=T#0.1S);
fbMonitor(fMinimumValidChange:=0.1, fMaximumFrameTime:=0.2);
AssertTrue(fbMonitor.bIsUpdating, Message:='Centroid update above threshold and is updating');

TEST_FINISHED();

TEST('Severity invalidation');

nCount := nCount + 1;
WriteCentroidValue(fbMonitor:=fbMonitor, fX:=0.0, fY:=0.0, nCount:=nCount, nX_Severity:=2, nY_Severity:=0, nCount_Severity:=0, tLastUpdate:=T#0.2S);
fbMonitor(fMinimumValidChange:=0.0);
AssertFalse(fbMonitor.bValid, Message:='Invalid data - x severity');

nCount := nCount + 1;
WriteCentroidValue(fbMonitor:=fbMonitor, fX:=0.1, fY:=0.1, nCount:=nCount, nX_Severity:=0, nY_Severity:=2, nCount_Severity:=0, tLastUpdate:=T#0.2S);
fbMonitor(fMinimumValidChange:=0.0);
AssertFalse(fbMonitor.bValid, Message:='Invalid data - y severity');

nCount := nCount + 1;
WriteCentroidValue(fbMonitor:=fbMonitor, fX:=0.2, fY:=0.2, nCount:=nCount, nX_Severity:=0, nY_Severity:=0, nCount_Severity:=2, tLastUpdate:=T#0.2S);
fbMonitor(fMinimumValidChange:=0.0);
AssertFalse(fbMonitor.bValid, Message:='Invalid data - count severity');

nCount := nCount + 1;
WriteCentroidValue(fbMonitor:=fbMonitor, fX:=0.0, fY:=0.0, nCount:=nCount, nX_Severity:=0, nY_Severity:=0, nCount_Severity:=0, tLastUpdate:=T#0.1S);
fbMonitor(fMinimumValidChange:=0.0);
AssertTrue(fbMonitor.bValid, Message:='Data valid');
AssertTrue(fbMonitor.bIsUpdating, Message:='Data valid and updating');

TEST_FINISHED();
END_METHOD

METHOD WriteCentroidValue
VAR_IN_OUT
    fbMonitor : FB_EpicsCentroidMonitor;
END_VAR
VAR_INPUT
    fX : LREAL;
    fY : LREAL;
    nCount : INT;
    nX_Severity : INT := 0;
    nY_Severity : INT := 0;
    nCount_Severity : INT := 0;
    tLastUpdate : TIME;
END_VAR
WRITE_PROTECTED_INT(ADR(fbMonitor.fbCentroidX.iPLCInternalSeverity), nX_Severity);
WRITE_PROTECTED_INT(ADR(fbMonitor.fbCentroidY.iPLCInternalSeverity), nY_Severity);
WRITE_PROTECTED_INT(ADR(fbMonitor.fbArrayCounter.iPLCInternalSeverity), nCount_Severity);

WRITE_PROTECTED_LREAL(ADR(fbMonitor.fbCentroidX.fPLCInternalValue), fX);
WRITE_PROTECTED_LREAL(ADR(fbMonitor.fbCentroidY.fPLCInternalValue), fY);
WRITE_PROTECTED_LREAL(ADR(fbMonitor.fbArrayCounter.fPLCInternalValue), INT_TO_LREAL(nCount));

WRITE_PROTECTED_TIME(ADR(fbMonitor.tLastUpdate), TIME() - tLastUpdate);
END_METHOD

END_FUNCTION_BLOCK

// POUs/Tests/FB_Test_EpicsMotorMonitor
{attribute 'call_after_init'}
FUNCTION_BLOCK FB_Test_EpicsMotorMonitor EXTENDS TcUnit.FB_TestSuite
VAR_INPUT
END_VAR
VAR_OUTPUT
END_VAR
VAR
END_VAR

TestBasics();

METHOD TestBasics
VAR_INPUT
END_VAR
VAR_INST
    fbMonitor : FB_EpicsMotorMonitor;
END_VAR
TEST('Basic');

WriteData(fbMonitor:=fbMonitor, fRBV:=0.0, nMoving:=0, nStatus:=0, nRBV_Severity:=0, nStatus_Severity:=0, nMoving_Severity:=0);
fbMonitor();
AssertTrue(fbMonitor.bValid, Message:='Data valid');

TEST_FINISHED();


TEST('Severities');

WriteData(fbMonitor:=fbMonitor, fRBV:=0.0, nMoving:=0, nStatus:=0, nRBV_Severity:=2, nStatus_Severity:=0, nMoving_Severity:=0);
fbMonitor();
AssertFalse(fbMonitor.bValid, Message:='Invalid RBV');

WriteData(fbMonitor:=fbMonitor, fRBV:=0.0, nMoving:=0, nStatus:=0, nRBV_Severity:=0, nStatus_Severity:=2, nMoving_Severity:=0);
fbMonitor();
AssertFalse(fbMonitor.bValid, Message:='Invalid status');

WriteData(fbMonitor:=fbMonitor, fRBV:=0.0, nMoving:=0, nStatus:=0, nRBV_Severity:=0, nStatus_Severity:=0, nMoving_Severity:=2);
fbMonitor();
AssertFalse(fbMonitor.bValid, Message:='Invalid moving');

WriteData(fbMonitor:=fbMonitor, fRBV:=0.0, nMoving:=0, nStatus:=0, nRBV_Severity:=0, nStatus_Severity:=0, nMoving_Severity:=0);
fbMonitor();
AssertTrue(fbMonitor.bValid, Message:='All valid');

TEST_FINISHED();

TEST('Moving');

WriteData(fbMonitor:=fbMonitor, fRBV:=0.0, nMoving:=0 (* DMOV *), nStatus:=0, nRBV_Severity:=0, nStatus_Severity:=0, nMoving_Severity:=0);
fbMonitor();
AssertTrue(fbMonitor.bIsMoving, Message:='Moving');

WriteData(fbMonitor:=fbMonitor, fRBV:=0.0, nMoving:=1 (* DMOV *), nStatus:=0, nRBV_Severity:=0, nStatus_Severity:=0, nMoving_Severity:=0);
fbMonitor();
AssertFalse(fbMonitor.bIsMoving, Message:='Not moving');

TEST_FINISHED();

TEST('Position');

WriteData(fbMonitor:=fbMonitor, fRBV:=10.0, nMoving:=0, nStatus:=0, nRBV_Severity:=0, nStatus_Severity:=0, nMoving_Severity:=0);
fbMonitor();
AssertEquals_LREAL(Actual:=fbMonitor.fPosition, Expected:=10.0, Delta:=0.1, Message:='Position 1 OK');

WriteData(fbMonitor:=fbMonitor, fRBV:=20.0, nMoving:=0, nStatus:=0, nRBV_Severity:=0, nStatus_Severity:=0, nMoving_Severity:=0);
fbMonitor();
AssertEquals_LREAL(Actual:=fbMonitor.fPosition, Expected:=20.0, Delta:=0.1, Message:='Position 2 OK');

TEST_FINISHED();

TEST('MSTA set');

WriteData(fbMonitor:=fbMonitor, fRBV:=0.0, nMoving:=0, nStatus:=16#0FFFF, nRBV_Severity:=0, nStatus_Severity:=0, nMoving_Severity:=0);
fbMonitor();

AssertTrue(fbMonitor.stMSTA.bPositiveDirection, Message:='bPositiveDirection True');
AssertTrue(fbMonitor.stMSTA.bDone, Message:='bDone True');
AssertTrue(fbMonitor.stMSTA.bPlusLimitSwitch, Message:='bPlusLimitSwitch True');
AssertTrue(fbMonitor.stMSTA.bHomeLimitSwitch, Message:='bHomeLimitSwitch True');
AssertTrue(fbMonitor.stMSTA.bUnused0, Message:='bUnused0 True');
AssertTrue(fbMonitor.stMSTA.bClosedLoop, Message:='bClosedLoop True');
AssertTrue(fbMonitor.stMSTA.bSlipStall, Message:='bSlipStall True');
AssertTrue(fbMonitor.stMSTA.bHome, Message:='bHome True');
AssertTrue(fbMonitor.stMSTA.bEncoderPresent, Message:='bEncoderPresent True');
AssertTrue(fbMonitor.stMSTA.bHardwareProblem, Message:='bHardwareProblem True');
AssertTrue(fbMonitor.stMSTA.bMoving, Message:='bMoving True');
AssertTrue(fbMonitor.stMSTA.bGainSupport, Message:='bGainSupport True');
AssertTrue(fbMonitor.stMSTA.bCommError, Message:='bCommError True');
AssertTrue(fbMonitor.stMSTA.bMinusLimitSwitch, Message:='bMinusLimitSwitch True');
AssertTrue(fbMonitor.stMSTA.bHomed, Message:='bHomed True');

TEST_FINISHED();


TEST('MSTA zero');

WriteData(fbMonitor:=fbMonitor, fRBV:=0.0, nMoving:=0, nStatus:=16#0000, nRBV_Severity:=0, nStatus_Severity:=0, nMoving_Severity:=0);
fbMonitor();

AssertFalse(fbMonitor.stMSTA.bPositiveDirection, Message:='bPositiveDirection False');
AssertFalse(fbMonitor.stMSTA.bDone, Message:='bDone False');
AssertFalse(fbMonitor.stMSTA.bPlusLimitSwitch, Message:='bPlusLimitSwitch False');
AssertFalse(fbMonitor.stMSTA.bHomeLimitSwitch, Message:='bHomeLimitSwitch False');
AssertFalse(fbMonitor.stMSTA.bUnused0, Message:='bUnused0 False');
AssertFalse(fbMonitor.stMSTA.bClosedLoop, Message:='bClosedLoop False');
AssertFalse(fbMonitor.stMSTA.bSlipStall, Message:='bSlipStall False');
AssertFalse(fbMonitor.stMSTA.bHome, Message:='bHome False');
AssertFalse(fbMonitor.stMSTA.bEncoderPresent, Message:='bEncoderPresent False');
AssertFalse(fbMonitor.stMSTA.bHardwareProblem, Message:='bHardwareProblem False');
AssertFalse(fbMonitor.stMSTA.bMoving, Message:='bMoving False');
AssertFalse(fbMonitor.stMSTA.bGainSupport, Message:='bGainSupport False');
AssertFalse(fbMonitor.stMSTA.bCommError, Message:='bCommError False');
AssertFalse(fbMonitor.stMSTA.bMinusLimitSwitch, Message:='bMinusLimitSwitch False');
AssertFalse(fbMonitor.stMSTA.bHomed, Message:='bHomed False');

TEST_FINISHED();


TEST('MSTA something');

WriteData(fbMonitor:=fbMonitor, fRBV:=0.0, nMoving:=0, nStatus:=2#0100_0011_0000_0110, nRBV_Severity:=0, nStatus_Severity:=0, nMoving_Severity:=0);
fbMonitor();

AssertFalse(fbMonitor.stMSTA.bPositiveDirection, Message:='bPositiveDirection');
AssertTrue(fbMonitor.stMSTA.bDone, Message:='bDone');
AssertTrue(fbMonitor.stMSTA.bPlusLimitSwitch, Message:='bPlusLimitSwitch');
AssertFalse(fbMonitor.stMSTA.bHomeLimitSwitch, Message:='bHomeLimitSwitch');

AssertFalse(fbMonitor.stMSTA.bUnused0, Message:='bUnused0');
AssertFalse(fbMonitor.stMSTA.bClosedLoop, Message:='bClosedLoop');
AssertFalse(fbMonitor.stMSTA.bSlipStall, Message:='bSlipStall');
AssertFalse(fbMonitor.stMSTA.bHome, Message:='bHome');

AssertTrue(fbMonitor.stMSTA.bEncoderPresent, Message:='bEncoderPresent');
AssertTrue(fbMonitor.stMSTA.bHardwareProblem, Message:='bHardwareProblem');
AssertFalse(fbMonitor.stMSTA.bMoving, Message:='bMoving');
AssertFalse(fbMonitor.stMSTA.bGainSupport, Message:='bGainSupport');

AssertFalse(fbMonitor.stMSTA.bCommError, Message:='bCommError');
AssertFalse(fbMonitor.stMSTA.bMinusLimitSwitch, Message:='bMinusLimitSwitch');
AssertTrue(fbMonitor.stMSTA.bHomed, Message:='bHomed');

TEST_FINISHED();
END_METHOD

METHOD WriteData
VAR_IN_OUT
    fbMonitor : FB_EpicsMotorMonitor;
END_VAR
VAR_INPUT
    fRBV : LREAL;
    nMoving : INT;
    nStatus : UINT;
    nRBV_Severity : INT := 0;
    nStatus_Severity : INT := 0;
    nMoving_Severity : INT := 0;
END_VAR
WRITE_PROTECTED_INT(ADR(fbMonitor.fbRBVCheck.iPLCInternalSeverity), nRBV_Severity);
WRITE_PROTECTED_INT(ADR(fbMonitor.fbMotorStatusCheck.iPLCInternalSeverity), nStatus_Severity);
WRITE_PROTECTED_INT(ADR(fbMonitor.fbMovingCheck.iPLCInternalSeverity), nMoving_Severity);

WRITE_PROTECTED_LREAL(ADR(fbMonitor.fbRBVCheck.fPLCInternalValue), fRBV);
WRITE_PROTECTED_LREAL(ADR(fbMonitor.fbMotorStatusCheck.fPLCInternalValue), UINT_TO_LREAL(nStatus));
WRITE_PROTECTED_LREAL(ADR(fbMonitor.fbMovingCheck.fPLCInternalValue), INT_TO_LREAL(nMoving));
END_METHOD

END_FUNCTION_BLOCK

// POUs/RUN_TESTS
PROGRAM RUN_TESTS
VAR
    // Logger
    {attribute 'analysis' := '-33'}
    fbCbTest : FB_CircuitBreaker_Test;
    {attribute 'analysis' := '-33'}
    // Data
    fbCentroidTest : FB_Test_EpicsCentroidMonitor;
    {attribute 'analysis' := '-33'}
    fbMotorTest : FB_Test_EpicsMotorMonitor;
    // EPS
    {attribute 'analysis' := '-33'}
    fbFlutterTest : FB_FlutterDetection_Test;
    // Hardware
    {attribute 'analysis' := '-33'}
    fbECATAutoRestartTest : FB_ECATAutoRestart_Test;
END_VAR

TcUnit.RUN();

END_PROGRAM
